// TIA Portal V21 export
VAR_GLOBAL   // PLC tag table "KAllComunicazione"
END_VAR
VAR_GLOBAL CONSTANT   // user constants
   KAllComun_PUT_Alarm : Int := 1;   // PUT_Alarm
   KAllComun_Get_Alarm : Int := 2;   // Get_Alarm
   KALLComunicazione_03 : Int := 3;
   KALLComunicazione_04 : Int := 4;
   KAllComun_Watchdog : Int := 5;   // Watchdog
   KALLComunicazione_06 : Int := 6;
   KALLComunicazione_07 : Int := 7;
   KALLComunicazione_08 : Int := 8;
   KALLComunicazione_09 : Int := 9;
   KALLComunicazione_10 : Int := 10;
   KALLComunicazione_11 : Int := 11;
   KALLComunicazione_12 : Int := 12;
   KALLComunicazione_13 : Int := 13;
   KALLComunicazione_14 : Int := 14;
   KALLComunicazione_15 : Int := 15;
   KALLComunicazione_16 : Int := 16;
END_VAR
